Staubli VAL3: pallet_getPos.pgx

program pallet_getPos(string x_sPalletName (dimensions=1), num& x_nPos (dimensions=1))
begin
  // get the actual position of the x_sPalletName
  call pallet:getPalletPos(x_sPalletName,x_nPos)
end
